// TIA Portal V21 export
FUNCTION "END PRINT" : Void   // FC19, LAD
{ S7_Optimized_Access := 'TRUE' }
// stored: SetENOAutomatically false
BEGIN

REGION Network 1: RECORD TIME
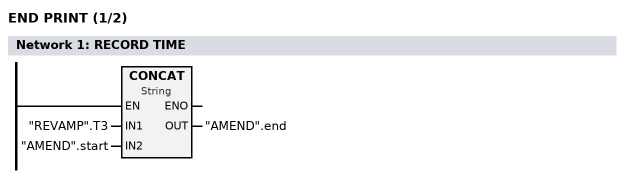
   RUNG wire#powerrail
      { S7_Templates := "[card := 2, str_type := String]" } CONCAT(IN1 := "REVAMP".T3, IN2 := "AMEND".start, OUT => "AMEND".end)
   END_RUNG
   // the same network as SCL:
   CONCAT(IN1 := "REVAMP".T3, IN2 := "AMEND".start, OUT => "AMEND".end);
END_REGION

REGION Network 2: PV CONCATE
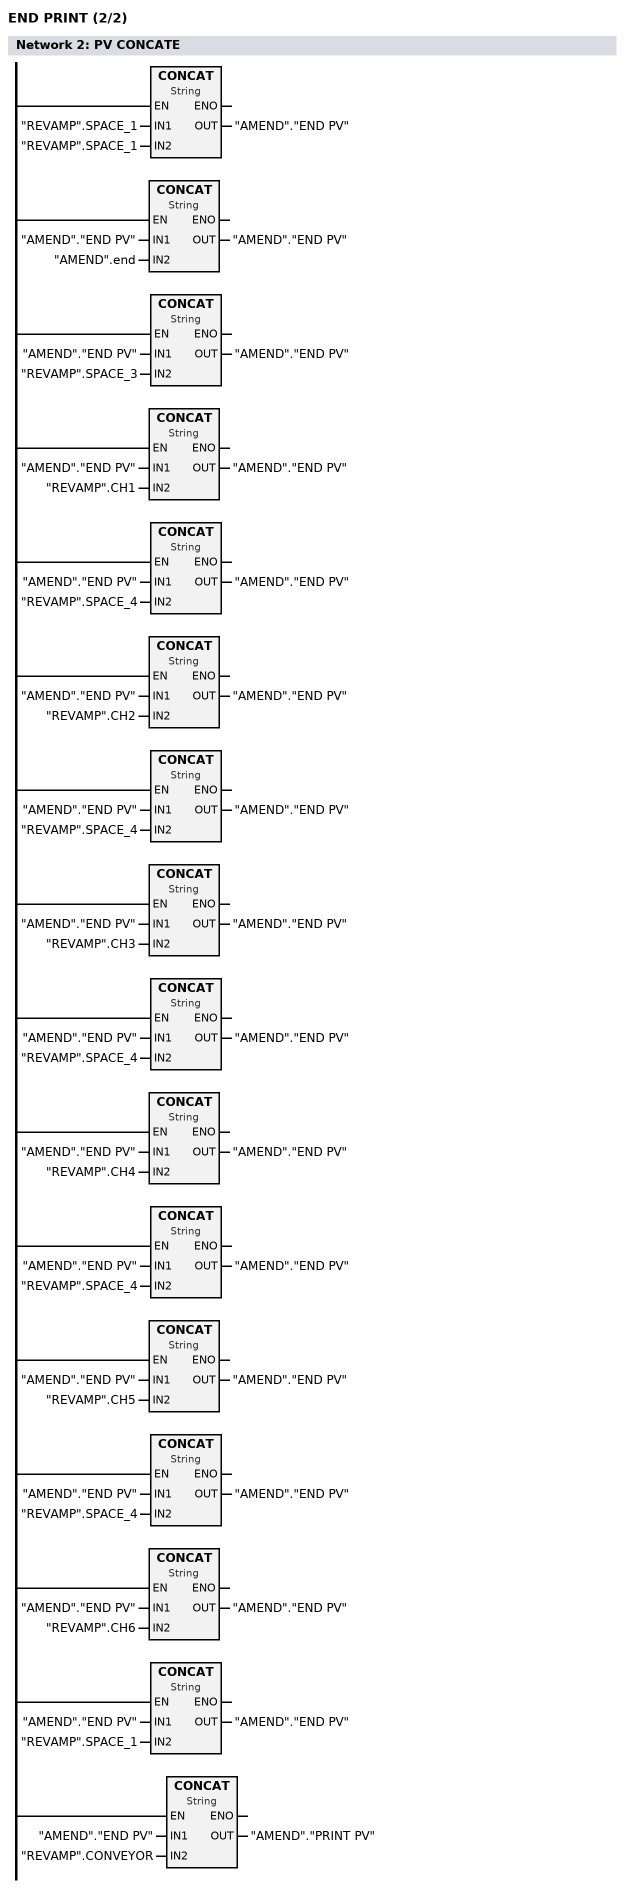
   RUNG wire#powerrail
      { S7_Templates := "[card := 2, str_type := String]" } CONCAT(IN1 := "REVAMP".SPACE_1, IN2 := "REVAMP".SPACE_1, OUT => "AMEND"."END PV")
   END_RUNG
   RUNG wire#powerrail
      { S7_Templates := "[card := 2, str_type := String]" } CONCAT(IN1 := "AMEND"."END PV", IN2 := "AMEND".end, OUT => "AMEND"."END PV")
   END_RUNG
   RUNG wire#powerrail
      { S7_Templates := "[card := 2, str_type := String]" } CONCAT(IN1 := "AMEND"."END PV", IN2 := "REVAMP".SPACE_3, OUT => "AMEND"."END PV")
   END_RUNG
   RUNG wire#powerrail
      { S7_Templates := "[card := 2, str_type := String]" } CONCAT(IN1 := "AMEND"."END PV", IN2 := "REVAMP".CH1, OUT => "AMEND"."END PV")
   END_RUNG
   RUNG wire#powerrail
      { S7_Templates := "[card := 2, str_type := String]" } CONCAT(IN1 := "AMEND"."END PV", IN2 := "REVAMP".SPACE_4, OUT => "AMEND"."END PV")
   END_RUNG
   RUNG wire#powerrail
      { S7_Templates := "[card := 2, str_type := String]" } CONCAT(IN1 := "AMEND"."END PV", IN2 := "REVAMP".CH2, OUT => "AMEND"."END PV")
   END_RUNG
   RUNG wire#powerrail
      { S7_Templates := "[card := 2, str_type := String]" } CONCAT(IN1 := "AMEND"."END PV", IN2 := "REVAMP".SPACE_4, OUT => "AMEND"."END PV")
   END_RUNG
   RUNG wire#powerrail
      { S7_Templates := "[card := 2, str_type := String]" } CONCAT(IN1 := "AMEND"."END PV", IN2 := "REVAMP".CH3, OUT => "AMEND"."END PV")
   END_RUNG
   RUNG wire#powerrail
      { S7_Templates := "[card := 2, str_type := String]" } CONCAT(IN1 := "AMEND"."END PV", IN2 := "REVAMP".SPACE_4, OUT => "AMEND"."END PV")
   END_RUNG
   RUNG wire#powerrail
      { S7_Templates := "[card := 2, str_type := String]" } CONCAT(IN1 := "AMEND"."END PV", IN2 := "REVAMP".CH4, OUT => "AMEND"."END PV")
   END_RUNG
   RUNG wire#powerrail
      { S7_Templates := "[card := 2, str_type := String]" } CONCAT(IN1 := "AMEND"."END PV", IN2 := "REVAMP".SPACE_4, OUT => "AMEND"."END PV")
   END_RUNG
   RUNG wire#powerrail
      { S7_Templates := "[card := 2, str_type := String]" } CONCAT(IN1 := "AMEND"."END PV", IN2 := "REVAMP".CH5, OUT => "AMEND"."END PV")
   END_RUNG
   RUNG wire#powerrail
      { S7_Templates := "[card := 2, str_type := String]" } CONCAT(IN1 := "AMEND"."END PV", IN2 := "REVAMP".SPACE_4, OUT => "AMEND"."END PV")
   END_RUNG
   RUNG wire#powerrail
      { S7_Templates := "[card := 2, str_type := String]" } CONCAT(IN1 := "AMEND"."END PV", IN2 := "REVAMP".CH6, OUT => "AMEND"."END PV")
   END_RUNG
   RUNG wire#powerrail
      { S7_Templates := "[card := 2, str_type := String]" } CONCAT(IN1 := "AMEND"."END PV", IN2 := "REVAMP".SPACE_1, OUT => "AMEND"."END PV")
   END_RUNG
   RUNG wire#powerrail
      { S7_Templates := "[card := 2, str_type := String]" } CONCAT(IN1 := "AMEND"."END PV", IN2 := "REVAMP".CONVEYOR, OUT => "AMEND"."PRINT PV")
   END_RUNG
   // the same network as SCL:
   CONCAT(IN1 := "REVAMP".SPACE_1, IN2 := "REVAMP".SPACE_1, OUT => "AMEND"."END PV");
   CONCAT(IN1 := "AMEND"."END PV", IN2 := "AMEND".end, OUT => "AMEND"."END PV");
   CONCAT(IN1 := "AMEND"."END PV", IN2 := "REVAMP".SPACE_3, OUT => "AMEND"."END PV");
   CONCAT(IN1 := "AMEND"."END PV", IN2 := "REVAMP".CH1, OUT => "AMEND"."END PV");
   CONCAT(IN1 := "AMEND"."END PV", IN2 := "REVAMP".SPACE_4, OUT => "AMEND"."END PV");
   CONCAT(IN1 := "AMEND"."END PV", IN2 := "REVAMP".CH2, OUT => "AMEND"."END PV");
   CONCAT(IN1 := "AMEND"."END PV", IN2 := "REVAMP".SPACE_4, OUT => "AMEND"."END PV");
   CONCAT(IN1 := "AMEND"."END PV", IN2 := "REVAMP".CH3, OUT => "AMEND"."END PV");
   CONCAT(IN1 := "AMEND"."END PV", IN2 := "REVAMP".SPACE_4, OUT => "AMEND"."END PV");
   CONCAT(IN1 := "AMEND"."END PV", IN2 := "REVAMP".CH4, OUT => "AMEND"."END PV");
   CONCAT(IN1 := "AMEND"."END PV", IN2 := "REVAMP".SPACE_4, OUT => "AMEND"."END PV");
   CONCAT(IN1 := "AMEND"."END PV", IN2 := "REVAMP".CH5, OUT => "AMEND"."END PV");
   CONCAT(IN1 := "AMEND"."END PV", IN2 := "REVAMP".SPACE_4, OUT => "AMEND"."END PV");
   CONCAT(IN1 := "AMEND"."END PV", IN2 := "REVAMP".CH6, OUT => "AMEND"."END PV");
   CONCAT(IN1 := "AMEND"."END PV", IN2 := "REVAMP".SPACE_1, OUT => "AMEND"."END PV");
   CONCAT(IN1 := "AMEND"."END PV", IN2 := "REVAMP".CONVEYOR, OUT => "AMEND"."PRINT PV");
END_REGION
END_FUNCTION
